ABB RAPID module: Module1.mod

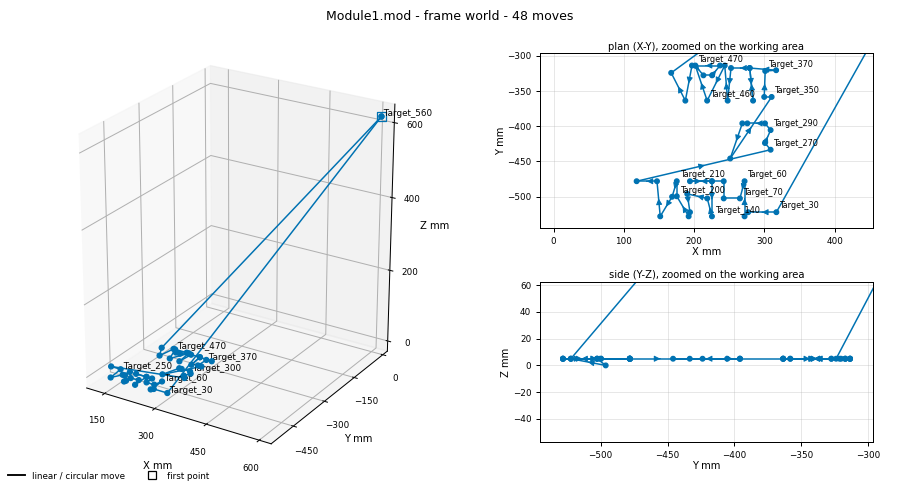
[picture p0: tool path of Module1.mod in frame world, 48 of 48 moves have a stored position in this frame; points joined in program order, loops and branches not executed]
MODULE Module1
        CONST robtarget Target_560:=[[610.214698352,0,619.499997666],[0.499999994,0,0.866025407,0],[0,0,0,0],[9E+09,9E+09,9E+09,9E+09,9E+09,9E+09]];
    CONST robtarget Target_30:=[[270.977,12.689,0],[0,0,1,0],[-1,0,-1,0],[9E+09,9E+09,9E+09,9E+09,9E+09,9E+09]];
    CONST robtarget Target_40:=[[230.782,12.689,0],[0,0,1,0],[0,0,0,0],[9E+09,9E+09,9E+09,9E+09,9E+09,9E+09]];
    CONST robtarget Target_50:=[[225.718,6.773,0],[0,0,1,0],[0,0,0,0],[9E+09,9E+09,9E+09,9E+09,9E+09,9E+09]];
    CONST robtarget Target_60:=[[225.718,56.773,0],[0,0,1,0],[0,0,0,0],[9E+09,9E+09,9E+09,9E+09,9E+09,9E+09]];
    CONST robtarget Target_70:=[[219.073,32.3,0],[0,0,1,0],[0,0,0,0],[9E+09,9E+09,9E+09,9E+09,9E+09,9E+09]];
    CONST robtarget Target_80:=[[196.058,32.3,0],[0,0,1,0],[0,0,0,0],[9E+09,9E+09,9E+09,9E+09,9E+09,9E+09]];
    CONST robtarget Target_100:=[[196.058,56.773,0],[0,0,1,0],[0,0,0,0],[9E+09,9E+09,9E+09,9E+09,9E+09,9E+09]];
    CONST robtarget Target_110:=[[179.283,56.773,0],[0,0,1,0],[0,0,0,0],[9E+09,9E+09,9E+09,9E+09,9E+09,9E+09]];
    CONST robtarget Target_120:=[[148.003,56.773,0],[0,0,1,0],[0,0,0,0],[9E+09,9E+09,9E+09,9E+09,9E+09,9E+09]];
    CONST robtarget Target_130:=[[179.283,56.773,0],[0,0,1,0],[0,0,0,0],[9E+09,9E+09,9E+09,9E+09,9E+09,9E+09]];
    CONST robtarget Target_140:=[[179.283,6.773,0],[0,0,1,0],[0,0,0,0],[9E+09,9E+09,9E+09,9E+09,9E+09,9E+09]];
    CONST robtarget Target_150:=[[172.638,32.3,0],[0,0,1,0],[0,0,0,0],[9E+09,9E+09,9E+09,9E+09,9E+09,9E+09]];
    CONST robtarget Target_160:=[[144.139,38.729,-5],[0,0,1,0],[0,0,0,0],[9E+09,9E+09,9E+09,9E+09,9E+09,9E+09]];
    CONST robtarget Target_180:=[[148.003,12.689,0],[0,0,1,0],[0,0,0,0],[9E+09,9E+09,9E+09,9E+09,9E+09,9E+09]];
    CONST robtarget Target_190:=[[146.139,6.773,0],[0,0,1,0],[0,0,0,0],[9E+09,9E+09,9E+09,9E+09,9E+09,9E+09]];
    CONST robtarget Target_200:=[[129.243,35.339,0],[0,0,1,0],[0,0,0,0],[9E+09,9E+09,9E+09,9E+09,9E+09,9E+09]];
    CONST robtarget Target_210:=[[129.243,56.773,0],[0,0,1,0],[0,0,0,0],[9E+09,9E+09,9E+09,9E+09,9E+09,9E+09]];
    CONST robtarget Target_220:=[[122.598,34.65,0],[0,0,1,0],[0,0,0,0],[9E+09,9E+09,9E+09,9E+09,9E+09,9E+09]];
    CONST robtarget Target_230:=[[105.701,6.773,0],[0,0,1,0],[0,0,0,0],[9E+09,9E+09,9E+09,9E+09,9E+09,9E+09]];
    CONST robtarget Target_250:=[[101.082,56.773,0],[0,0,1,0],[0,0,0,0],[9E+09,9E+09,9E+09,9E+09,9E+09,9E+09]];
    CONST robtarget Target_260:=[[72.111,56.773,0],[0,0,1,0],[0,0,0,0],[9E+09,9E+09,9E+09,9E+09,9E+09,9E+09]];
    CONST robtarget Target_270:=[[262.792,101.577,0],[0,0,1,0],[0,0,0,0],[9E+09,9E+09,9E+09,9E+09,9E+09,9E+09]];
    CONST robtarget Target_280:=[[254.769,111.139,0],[0,0,1,0],[0,0,0,0],[9E+09,9E+09,9E+09,9E+09,9E+09,9E+09]];
    CONST robtarget Target_290:=[[262.792,129.534,0],[0,0,1,0],[0,0,0,0],[9E+09,9E+09,9E+09,9E+09,9E+09,9E+09]];
    CONST robtarget Target_300:=[[254.769,139.097,0],[0,0,1,0],[0,0,0,0],[9E+09,9E+09,9E+09,9E+09,9E+09,9E+09]];
    CONST robtarget Target_320:=[[229.688,139.097,0],[0,0,1,0],[0,0,0,0],[9E+09,9E+09,9E+09,9E+09,9E+09,9E+09]];
    CONST robtarget Target_330:=[[222.517,139.097,0],[0,0,1,0],[0,0,0,0],[9E+09,9E+09,9E+09,9E+09,9E+09,9E+09]];
    CONST robtarget Target_340:=[[205.296,89.097,0],[0,0,1,0],[0,0,0,0],[9E+09,9E+09,9E+09,9E+09,9E+09,9E+09]];
    CONST robtarget Target_350:=[[264.251,176.729,0],[0,0,1,0],[0,0,0,0],[9E+09,9E+09,9E+09,9E+09,9E+09,9E+09]];
    CONST robtarget Target_360:=[[253.675,176.729,0],[0,0,1,0],[0,0,0,0],[9E+09,9E+09,9E+09,9E+09,9E+09,9E+09]];
    CONST robtarget Target_370:=[[255.094,213.641,0],[0,0,1,0],[0,0,0,0],[9E+09,9E+09,9E+09,9E+09,9E+09,9E+09]];
    CONST robtarget Target_380:=[[270.653,214.735,0],[0,0,1,0],[0,0,0,0],[9E+09,9E+09,9E+09,9E+09,9E+09,9E+09]];
    CONST robtarget Target_390:=[[233.051,217.855,0],[0,0,1,0],[0,0,0,0],[9E+09,9E+09,9E+09,9E+09,9E+09,9E+09]];
    CONST robtarget Target_400:=[[237.833,171.421,0],[0,0,1,0],[0,0,0,0],[9E+09,9E+09,9E+09,9E+09,9E+09,9E+09]];
    CONST robtarget Target_410:=[[233.051,217.855,0],[0,0,1,0],[0,0,0,0],[9E+09,9E+09,9E+09,9E+09,9E+09,9E+09]];
    CONST robtarget Target_420:=[[206.431,217.855,0],[0,0,1,0],[0,0,0,0],[9E+09,9E+09,9E+09,9E+09,9E+09,9E+09]];
    CONST robtarget Target_430:=[[201.65,171.421,0],[0,0,1,0],[0,0,0,0],[9E+09,9E+09,9E+09,9E+09,9E+09,9E+09]];
    CONST robtarget Target_440:=[[197.517,221.421,0],[0,0,1,0],[0,0,0,0],[9E+09,9E+09,9E+09,9E+09,9E+09,9E+09]];
    CONST robtarget Target_460:=[[172.476,171.421,0],[0,0,1,0],[0,0,0,0],[9E+09,9E+09,9E+09,9E+09,9E+09,9E+09]];
    CONST robtarget Target_470:=[[155.62,221.421,0],[0,0,1,0],[0,0,0,0],[9E+09,9E+09,9E+09,9E+09,9E+09,9E+09]];
    CONST robtarget Target_480:=[[167.168,207.442,0],[0,0,1,0],[0,0,0,0],[9E+09,9E+09,9E+09,9E+09,9E+09,9E+09]];
    CONST robtarget Target_490:=[[179.501,207.442,0],[0,0,1,0],[0,0,0,0],[9E+09,9E+09,9E+09,9E+09,9E+09,9E+09]];
    CONST robtarget Target_500:=[[190.791,221.421,0],[0,0,1,0],[0,0,0,0],[9E+09,9E+09,9E+09,9E+09,9E+09,9E+09]];
    CONST robtarget Target_510:=[[150.88,221.421,0],[0,0,1,0],[0,0,0,0],[9E+09,9E+09,9E+09,9E+09,9E+09,9E+09]];
    CONST robtarget Target_530:=[[141.439,171.421,0],[0,0,1,0],[0,0,0,0],[9E+09,9E+09,9E+09,9E+09,9E+09,9E+09]];
    CONST robtarget Target_540:=[[121.301,211.007,0],[0,0,1,0],[0,0,0,0],[9E+09,9E+09,9E+09,9E+09,9E+09,9E+09]];
!***********************************************************
    !
    ! Module:  Module1
    !
    ! Description:
    !   <Insert description here>
    !
    ! Author: User
    !
    ! Version: 1.0
    !
    !***********************************************************


    !***********************************************************
    !
    ! Procedure main
    !
    !   This is the entry point of your program
    !
    !***********************************************************
    PROC main()
        !Add your code here
    ENDPROC
    PROC Path_10()
        MoveL Target_560,v1000,z100,marcadorf\WObj:=wobj0;
        MoveL Target_30,v1000,z100,marcadorf\WObj:=tablerof;
        MoveL Target_40,v1000,z100,marcadorf\WObj:=tablerof;
        MoveL Target_50,v1000,z100,marcadorf\WObj:=tablerof;
        MoveL Target_60,v1000,z100,marcadorf\WObj:=tablerof;
        MoveL Target_70,v1000,z100,marcadorf\WObj:=tablerof;
        MoveL Target_80,v1000,z100,marcadorf\WObj:=tablerof;
        MoveL Target_100,v1000,z100,marcadorf\WObj:=tablerof;
        MoveL Target_110,v1000,z100,marcadorf\WObj:=tablerof;
        MoveL Target_120,v1000,z100,marcadorf\WObj:=tablerof;
        MoveL Target_130,v1000,z100,marcadorf\WObj:=tablerof;
        MoveL Target_140,v1000,z100,marcadorf\WObj:=tablerof;
        MoveL Target_150,v1000,z100,marcadorf\WObj:=tablerof;
        MoveL Target_160,v1000,z100,marcadorf\WObj:=tablerof;
        MoveL Target_180,v1000,z100,marcadorf\WObj:=tablerof;
        MoveL Target_190,v1000,z100,marcadorf\WObj:=tablerof;
        MoveL Target_200,v1000,z100,marcadorf\WObj:=tablerof;
        MoveL Target_210,v1000,z100,marcadorf\WObj:=tablerof;
        MoveL Target_220,v1000,z100,marcadorf\WObj:=tablerof;
        MoveL Target_230,v1000,z100,marcadorf\WObj:=tablerof;
        MoveL Target_250,v1000,z100,marcadorf\WObj:=tablerof;
        MoveL Target_260,v1000,z100,marcadorf\WObj:=tablerof;
        MoveL Target_270,v1000,z100,marcadorf\WObj:=tablerof;
        MoveL Target_280,v1000,z100,marcadorf\WObj:=tablerof;
        MoveL Target_290,v1000,z100,marcadorf\WObj:=tablerof;
        MoveL Target_300,v1000,z100,marcadorf\WObj:=tablerof;
        MoveL Target_320,v1000,z100,marcadorf\WObj:=tablerof;
        MoveL Target_330,v1000,z100,marcadorf\WObj:=tablerof;
        MoveL Target_340,v1000,z100,marcadorf\WObj:=tablerof;
        MoveL Target_350,v1000,z100,marcadorf\WObj:=tablerof;
        MoveL Target_360,v1000,z100,marcadorf\WObj:=tablerof;
        MoveL Target_370,v1000,z100,marcadorf\WObj:=tablerof;
        MoveL Target_380,v1000,z100,marcadorf\WObj:=tablerof;
        MoveL Target_390,v1000,z100,marcadorf\WObj:=tablerof;
        MoveL Target_400,v1000,z100,marcadorf\WObj:=tablerof;
        MoveL Target_410,v1000,z100,marcadorf\WObj:=tablerof;
        MoveL Target_420,v1000,z100,marcadorf\WObj:=tablerof;
        MoveL Target_430,v1000,z100,marcadorf\WObj:=tablerof;
        MoveL Target_440,v1000,z100,marcadorf\WObj:=tablerof;
        MoveL Target_460,v1000,z100,marcadorf\WObj:=tablerof;
        MoveL Target_470,v1000,z100,marcadorf\WObj:=tablerof;
        MoveL Target_480,v1000,z100,marcadorf\WObj:=tablerof;
        MoveL Target_490,v1000,z100,marcadorf\WObj:=tablerof;
        MoveL Target_500,v1000,z100,marcadorf\WObj:=tablerof;
        MoveL Target_510,v1000,z100,marcadorf\WObj:=tablerof;
        MoveL Target_530,v1000,z100,marcadorf\WObj:=tablerof;
        MoveL Target_540,v1000,z100,marcadorf\WObj:=tablerof;
        MoveL Target_560,v1000,z100,marcadorf\WObj:=wobj0;
    ENDPROC
ENDMODULE
